// LS Electric XG5000 project: xg
// PLC LSPLC
// module base 0 slot 0: 입출력 모듈:XBC-DR32H (DC 24V 입력, 릴레이 출력 32점)
// module base 0 slot 1: 위치결정 모듈:XBF-PD02A (위치결정 펄스(LD)출력형, 2축)
// module base 0 slot 2: 출력 모듈:XBE-TN/TP16A (트랜지스터 출력, 16점 (싱크출력/소스출력))

PROGRAM NewProgram (task: 스캔 프로그램)

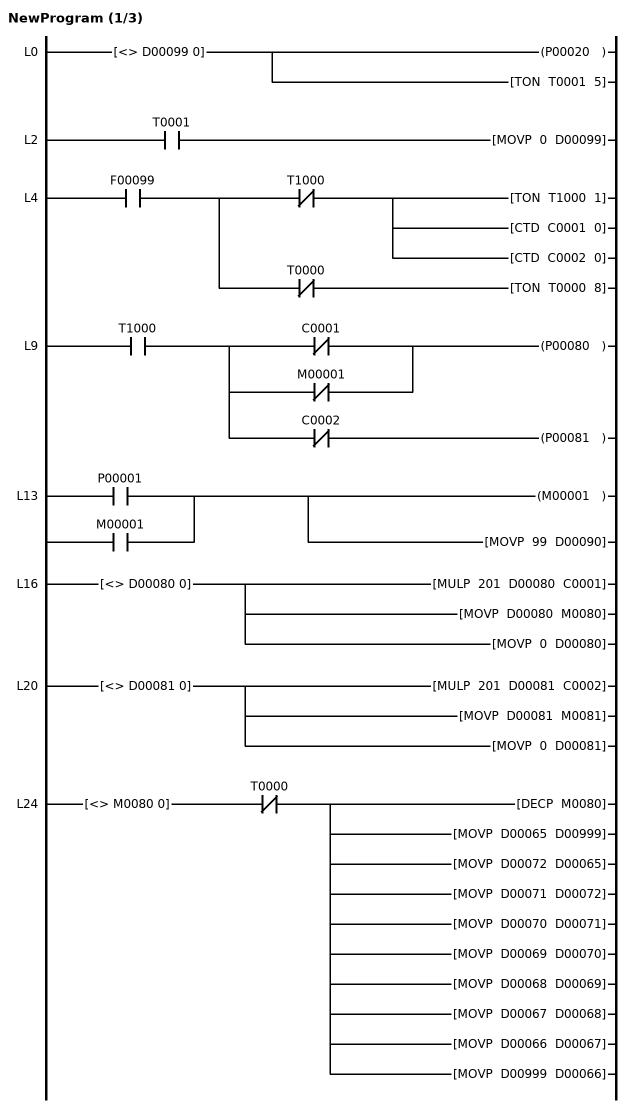
; L0
LOAD<>    D00099 0
OUT       P00020
TON       T0001 5
; L2
LOAD      T0001
MOVP      0 D00099
; L4
LOAD      F00099
MPUSH
AND NOT   T1000
TON       T1000 1
CTD       C0001 0
CTD       C0002 0
MPOP
AND NOT   T0000
TON       T0000 8
; L9
LOAD      T1000
MPUSH
LOAD NOT  C0001
OR NOT    M00001
AND LOAD
OUT       P00080
MPOP
AND NOT   C0002
OUT       P00081
; L13
LOAD      P00001
OR        M00001
OUT       M00001
MOVP      99 D00090
; L16
LOAD<>    D00080 0
MULP      201 D00080 C0001
MOVP      D00080 M0080
MOVP      0 D00080
; L20
LOAD<>    D00081 0
MULP      201 D00081 C0002
MOVP      D00081 M0081
MOVP      0 D00081
; L24
LOAD<>    M0080 0
AND NOT   T0000
DECP      M0080
MOVP      D00065 D00999
MOVP      D00072 D00065
MOVP      D00071 D00072
MOVP      D00070 D00071
MOVP      D00069 D00070
MOVP      D00068 D00069
MOVP      D00067 D00068
MOVP      D00066 D00067
MOVP      D00999 D00066

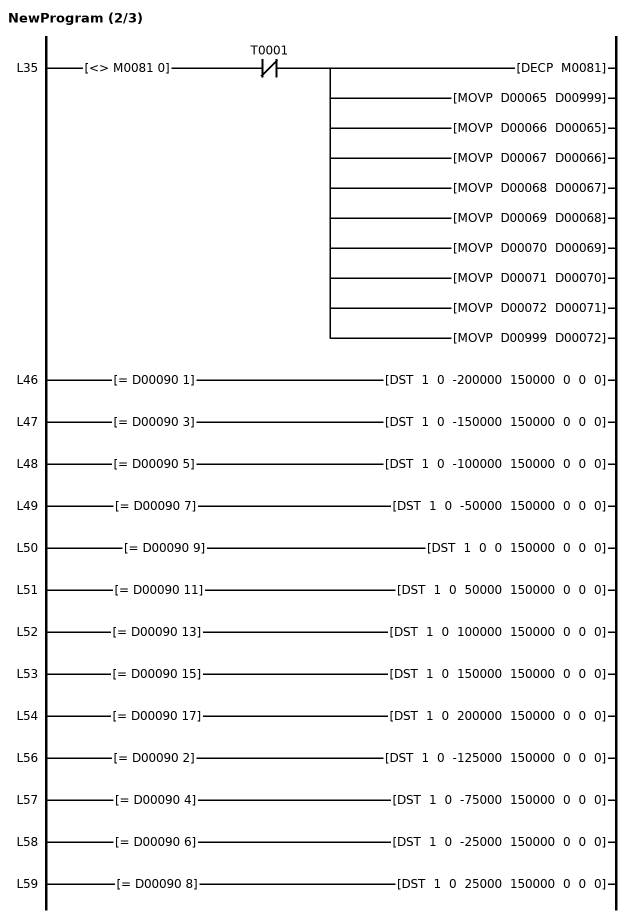
; L35
LOAD<>    M0081 0
AND NOT   T0001
DECP      M0081
MOVP      D00065 D00999
MOVP      D00066 D00065
MOVP      D00067 D00066
MOVP      D00068 D00067
MOVP      D00069 D00068
MOVP      D00070 D00069
MOVP      D00071 D00070
MOVP      D00072 D00071
MOVP      D00999 D00072
; L46
LOAD=     D00090 1
DST       1 0 -200000 150000 0 0 0
; L47
LOAD=     D00090 3
DST       1 0 -150000 150000 0 0 0
; L48
LOAD=     D00090 5
DST       1 0 -100000 150000 0 0 0
; L49
LOAD=     D00090 7
DST       1 0 -50000 150000 0 0 0
; L50
LOAD=     D00090 9
DST       1 0 0 150000 0 0 0
; L51
LOAD=     D00090 11
DST       1 0 50000 150000 0 0 0
; L52
LOAD=     D00090 13
DST       1 0 100000 150000 0 0 0
; L53
LOAD=     D00090 15
DST       1 0 150000 150000 0 0 0
; L54
LOAD=     D00090 17
DST       1 0 200000 150000 0 0 0
; L56
LOAD=     D00090 2
DST       1 0 -125000 150000 0 0 0
; L57
LOAD=     D00090 4
DST       1 0 -75000 150000 0 0 0
; L58
LOAD=     D00090 6
DST       1 0 -25000 150000 0 0 0
; L59
LOAD=     D00090 8
DST       1 0 25000 150000 0 0 0

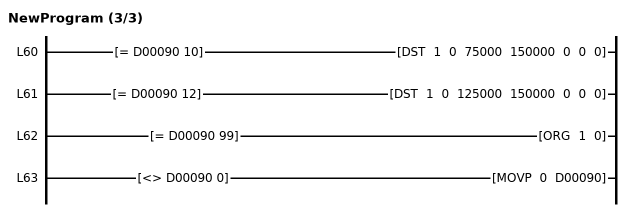
; L60
LOAD=     D00090 10
DST       1 0 75000 150000 0 0 0
; L61
LOAD=     D00090 12
DST       1 0 125000 150000 0 0 0
; L62
LOAD=     D00090 99
ORG       1 0
; L63
LOAD<>    D00090 0
MOVP      0 D00090